Fanuc KAREL source: kt00557.KL

-- PROVISIONAL review KL for V1013-1; original PC SHA256 924807e8fa6ade4dd3481606a2e377d5f31f71f4e71504275418cd2266f30981
-- Incomplete behavior may be omitted. Consult companion uncertainty JSON. Do not deploy.
PROGRAM KT00557
%NOLOCKGROUP
-- UNRESOLVED_DECL V1 type=000013
-- UNRESOLVED_DECL V2 type=000013
-- UNRESOLVED_DECL OUT type=000013
BEGIN
  -- UNRESOLVED_PC offsets 5-20; opcodes 2E,22,32,35
  -- UNRESOLVED_PC offsets 25-40; opcodes 2E,22,32,35
  -- UNRESOLVED_PC offsets 45-60; opcodes 2E,22,32,35
  -- UNRESOLVED_PC offsets 65-80; opcodes 2E,22,32,35
  -- UNRESOLVED_PC offsets 85-109; opcodes 49,49,93,4A
  -- UNRESOLVED_PC offsets 114-118; opcodes 7F
END KT00557
